INTERFACE I_PtTimesource

METHOD getDateTime : PtDateTime
VAR_INPUT
END_VAR
END_METHOD

END_INTERFACE

(* stored: Version 1.1.0.1, ProductVersion 3.1.4024.12
   Itf I_PtTimesource: Id {33c42691-f817-44a1-812e-0a01ddb29226}
   Method getDateTime: Id {893cc845-c23c-423d-9f71-b9d37c1869c5} *)
